// TIA Portal V17 export
// export: Created 2024-08-20T10:59:41.9879963Z, ExportSetting WithDefaults, DisplayName Totally Integrated Automation Portal, DisplayVersion V17 Update 4, DisplayName TIA Portal Openness, DisplayVersion V17 Update 4, DisplayName TIA Portal Version Control Interface, DisplayVersion V17, DisplayName STEP 7 Professional, DisplayVersion V17 Update 4, DisplayName STEP 7 Safety, DisplayVersion V17, DisplayName WinCC Advanced, DisplayVersion V17 Update 4
DATA_BLOCK "COMANDOS"   // DB303
{ S7_Optimized_Access := 'FALSE' }
VERSION : 0.1
// stored: AutoNumber false, DBAccessibleFromOPCUA true, IsOnlyStoredInLoadMemory false, IsWriteProtectedInAS false
   VAR RETAIN
      "MB-01-HS9" : Bool := false;   // Comando disponível
      "MB-01-HS10" : Bool := false;   // Comando disponível
      "MB-01-HS11" : Bool;   // Comando disponível
      "MB-01-HS12" : Bool;   // Comando disponível
      "MB-01-HS13" : Bool;   // Comando disponível
      "MB-01-HS14" : Bool;   // Comando disponível
      "MB-01-HS15" : Bool;   // Comando disponível
      "MB-01-HS16" : Bool;   // Comando disponível
      "MB-01-HS1" : Bool := true;   // Comando manual/automático
      "MB-01-HS2" : Bool := false;   // Comando liga
      "MB-01-HS3" : Bool := false;   // Comando desliga
      "MB-01-HS4" : Bool := false;   // Comando reset falha
      "MB-01-HS5" : Bool := false;   // Comando reset tempo de operação
      "MB-01-HS6" : Bool;
      "MB-01-HS7" : Bool := false;   // Comando habilita bloqueio
      "MB-01-HS8" : Bool := false;   // Comando disponível
      "MB-02-HS9" : Bool := false;   // Comando disponível
      "MB-02-HS10" : Bool := false;   // Comando disponível
      "MB-02-HS11" : Bool;   // Comando disponível
      "MB-02-HS12" : Bool;   // Comando disponível
      "MB-02-HS13" : Bool;   // Comando disponível
      "MB-02-HS14" : Bool;   // Comando disponível
      "MB-02-HS15" : Bool;   // Comando disponível
      "MB-02-HS16" : Bool;   // Comando disponível
      "MB-02-HS1" : Bool := true;   // Comando manual/automático
      "MB-02-HS2" : Bool := false;   // Comando liga
      "MB-02-HS3" : Bool := false;   // Comando desliga
      "MB-02-HS4" : Bool := false;   // Comando reset falha
      "MB-02-HS5" : Bool := false;   // Comando reset tempo de operação
      "MB-02-HS6" : Bool;
      "MB-02-HS7" : Bool := false;   // Comando habilita bloqueio
      "MB-02-HS8" : Bool := false;   // Comando disponível
      "MB-03-HS9" : Bool := false;   // Comando disponível
      "MB-03-HS10" : Bool := false;   // Comando disponível
      "MB-03-HS11" : Bool;   // Comando disponível
      "MB-03-HS12" : Bool;   // Comando disponível
      "MB-03-HS13" : Bool;   // Comando disponível
      "MB-03-HS14" : Bool;   // Comando disponível
      "MB-03-HS15" : Bool;   // Comando disponível
      "MB-03-HS16" : Bool;   // Comando disponível
      "MB-03-HS1" : Bool := true;   // Comando manual/automático
      "MB-03-HS2" : Bool := false;   // Comando liga
      "MB-03-HS3" : Bool := false;   // Comando desliga
      "MB-03-HS4" : Bool := false;   // Comando reset falha
      "MB-03-HS5" : Bool := false;   // Comando reset tempo de operação
      "MB-03-HS6" : Bool;
      "MB-03-HS7" : Bool := false;   // Comando habilita bloqueio
      "MB-03-HS8" : Bool := false;   // Comando disponível
      "MB-04-HS9" : Bool := false;   // Comando disponível
      "MB-04-HS10" : Bool := false;   // Comando disponível
      "MB-04-HS11" : Bool;   // Comando disponível
      "MB-04-HS12" : Bool;   // Comando disponível
      "MB-04-HS13" : Bool;   // Comando disponível
      "MB-04-HS14" : Bool;   // Comando disponível
      "MB-04-HS15" : Bool;   // Comando disponível
      "MB-04-HS16" : Bool;   // Comando disponível
      "MB-04-HS1" : Bool := false;   // Comando manual/automático
      "MB-04-HS2" : Bool := false;   // Comando liga
      "MB-04-HS3" : Bool := false;   // Comando desliga
      "MB-04-HS4" : Bool := false;   // Comando reset falha
      "MB-04-HS5" : Bool := false;   // Comando reset tempo de operação
      "MB-04-HS6" : Bool;
      "MB-04-HS7" : Bool := false;   // Comando habilita bloqueio
      "MB-04-HS8" : Bool := false;   // Comando disponível
      "LIT_001-HS9" : Bool;   // Comando disponível
      "LIT_001-HS10" : Bool;   // Comando disponível
      "LIT_001-HS11" : Bool;   // Comando disponível
      "LIT_001-HS12" : Bool;   // Comando disponível
      "LIT_001-HS13" : Bool;   // Comando disponível
      "LIT_001-HS14" : Bool;   // Comando disponível
      "LIT_001-HS15" : Bool;   // Comando disponível
      "LIT_001-HS16" : Bool;   // Comando disponível
      "LIT_001-HSHH" : Bool;   // Inibe alarme muito alto montante peneira 1
      "LIT_001-HSH" : Bool;   // Inibe alarme nível alto montante peneira 1
      "LIT_001-HSL" : Bool;   // Inibe alarme nível baixo montante peneira 1
      "LIT_001-HSLL" : Bool;   // Inibe alarme nível muito baixo montante peneira 1
      "LIT_001-HSM" : Bool;   // Habilita valor manual para medidor
      "LIT_001-HS6" : Bool;   // Comando disponível
      "LIT_001-HS7" : Bool;   // Comando disponível
      "LIT_001-HS8" : Bool;   // Comando disponível
      "PID-TA3-HI" : Bool;   // Habilita integrall PID tanque de aeração
      "PID-EEEB-HD" : Bool;   // Habilita derivativo PID tanque de aeração
      "PID-EEEB-HP" : Bool;   // Habilita proporcional PID tanque de aeração
      "PID-EEEB-HI" : Bool;   // Habilita integrall PID tanque de aeração
      "PID-TA5-HD" : Bool;   // Habilita derivativo PID tanque de aeração
      "PID-TA5-HP" : Bool;   // Habilita proporcional PID tanque de aeração
      "PID-TA5-HI" : Bool;   // Habilita integrall PID tanque de aeração
      "PID-TA1-HM" : Bool;   // Habilita valor manual para saída
      "PID-TA1-HD" : Bool;   // Habilita derivativo PID tanque de aeração
      "PID-TA1-HP" : Bool;   // Habilita proporcional PID tanque de aeração
      "PID-TA1-HI" : Bool;   // Habilita integrall PID tanque de aeração
      "PID-TA2-HD" : Bool;   // Habilita derivativo PID tanque de aeração
      "PID-TA2-HP" : Bool;   // Habilita proporcional PID tanque de aeração
      "PID-TA2-HI" : Bool;   // Habilita integrall PID tanque de aeração
      "PID-TA3-HD" : Bool;   // Habilita derivativo PID tanque de aeração
      "PID-TA3-HP" : Bool;   // Habilita proporcional PID tanque de aeração
      "PID-TA2-HM" : Bool;   // Habilita valor manual para saída
      "PID-TA3-HM" : Bool;   // Habilita valor manual para saída
      "PID-EEEB-HM" : Bool;   // Habilita valor manual para saída
      "PID-TA5-HM" : Bool;   // Habilita valor manual para saída
   END_VAR
BEGIN
END_DATA_BLOCK
